TYPE StartupFanDelay :
STRUCT
	SupplyFan: LTIME;
	ExtractFan: LTIME;
END_STRUCT
END_TYPE

(* stored: Version 1.1.0.1, ProductVersion 3.1.4024.6
   DUT StartupFanDelay: Id {cec732d7-d442-4ea9-bf62-be87ed57bf62} *)
